// TIA Portal V18 export
DATA_BLOCK "CMMS_Z1_FHPP_DPWR_DAT_DB"   // DB71
AUTHOR : FESTO
FAMILY : E-DRIVE
VERSION : 5.1
// stored: AutoNumber true, DBAccessibleFromOPCUA true, InstanceOfName FHPP_DPWR_DAT, InstanceOfType FB
"FHPP_DPWR_DAT"
   // VAR_INPUT
   //    HW_IO_FHPP : HW_IO;
   //    HW_IO_FPC : HW_IO;
   //    HW_IO_FHPPplus : HW_IO;
   //    cfgFHPPplusOut : DInt;
   // END_VAR
   // VAR_OUTPUT
   //    Error : Bool;
   //    Status : "DT_FML_STATUS";
   // END_VAR
   // VAR_IN_OUT
   //    FML_REF : "DT_FML_REF";
   // END_VAR
   // VAR
   //    EnableFHPPplusOutOld : DInt;
   //    FHPPplusSize { ExternalAccessible := 'False'; ExternalVisible := 'False'; ExternalWritable := 'False'} : DInt;
   //    FHPPplusElementSize { ExternalAccessible := 'False'; ExternalVisible := 'False'; ExternalWritable := 'False'} : Array[1..9] of DInt;
   // END_VAR
BEGIN
END_DATA_BLOCK
